FUNCTION_BLOCK FB_Observer_LINT EXTENDS FB_AbstractObserver
VAR
    _nVal:              LINT;
END_VAR

METHOD FB_init : BOOL
VAR_INPUT
	bInitRetains : BOOL; // if TRUE, the retain variables are initialized (warm start / cold start)
	bInCopyCode : BOOL;  // if TRUE, the instance afterwards gets moved into the copy code (online change)
END_VAR
THIS^._nTypeClass := __SYSTEM.TYPE_CLASS.TYPE_LINT;
THIS^._pVal := ADR(THIS^._nVal);
THIS^._nSize := SIZEOF(THIS^._nVal);
END_METHOD

PROPERTY nValue64 : LINT
GET
nValue64 := THIS^._nVal;
END_GET
END_PROPERTY

END_FUNCTION_BLOCK

(* stored: Version 1.1.0.1, ProductVersion 3.1.4024.12
   POU FB_Observer_LINT: Id {7cc927c9-1c83-07c4-350d-bb0574d22968}, SpecialFunc None
   Method FB_init: Id {f6e00212-579e-00a0-2bda-1ffeeb4a1c1c}
   Property nValue64: Id {87ea8490-b7d8-0abd-12c0-3ae03fa02b22}
   Get Get: Id {d4ec44b2-0d19-09c0-123e-f4610ba9ee04} *)
